DATA_BLOCK "DB_HVAC_IO"
{ S7_Optimized_Access := 'FALSE' }
VERSION : 1.0
   STRUCT
      Data : "UDT_HVAC_IO";
   END_STRUCT;
BEGIN
   Data.UseSimulation := TRUE;
END_DATA_BLOCK
